// Mitsubishi GX Works2 project: 20151109(M60~65変える前)   PLC: Q03UDV

PROGRAM P1
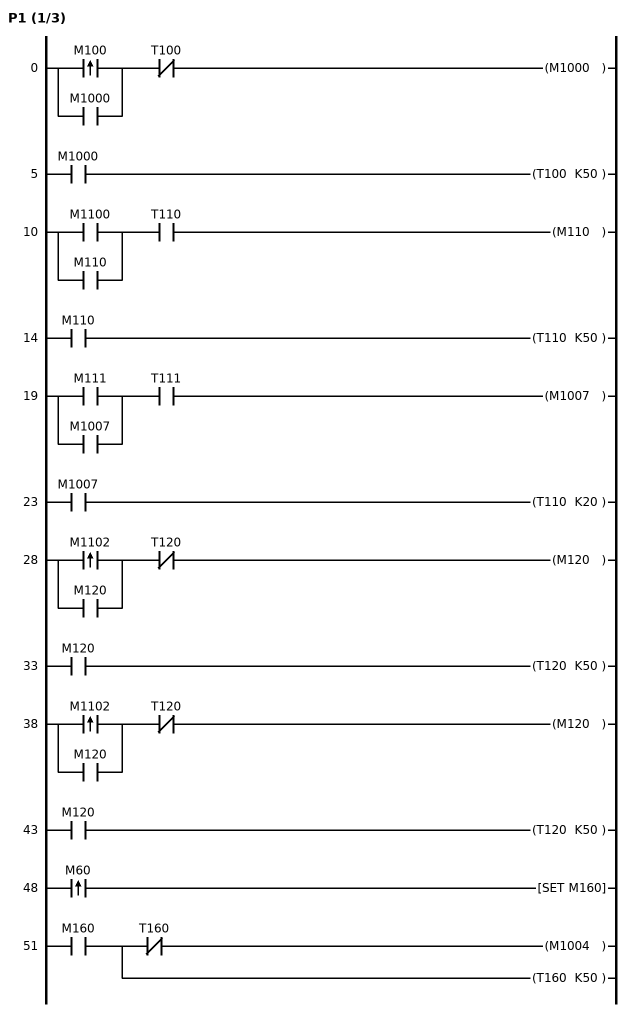
0     LDP     M100
      OR      M1000
      ANI     T100
      OUT     M1000
5     LD      M1000
      OUT     T100 K50
10    LD      M1100
      OR      M110
      AND     T110
      OUT     M110
14    LD      M110
      OUT     T110 K50
19    LD      M111
      OR      M1007
      AND     T111
      OUT     M1007
23    LD      M1007
      OUT     T110 K20
28    LDP     M1102
      OR      M120
      ANI     T120
      OUT     M120
33    LD      M120
      OUT     T120 K50
38    LDP     M1102
      OR      M120
      ANI     T120
      OUT     M120
43    LD      M120
      OUT     T120 K50
48    LDP     M60
      SET     M160
51    LD      M160
      MPS
      ANI     T160
      OUT     M1004
      MPP
      OUT     T160 K50
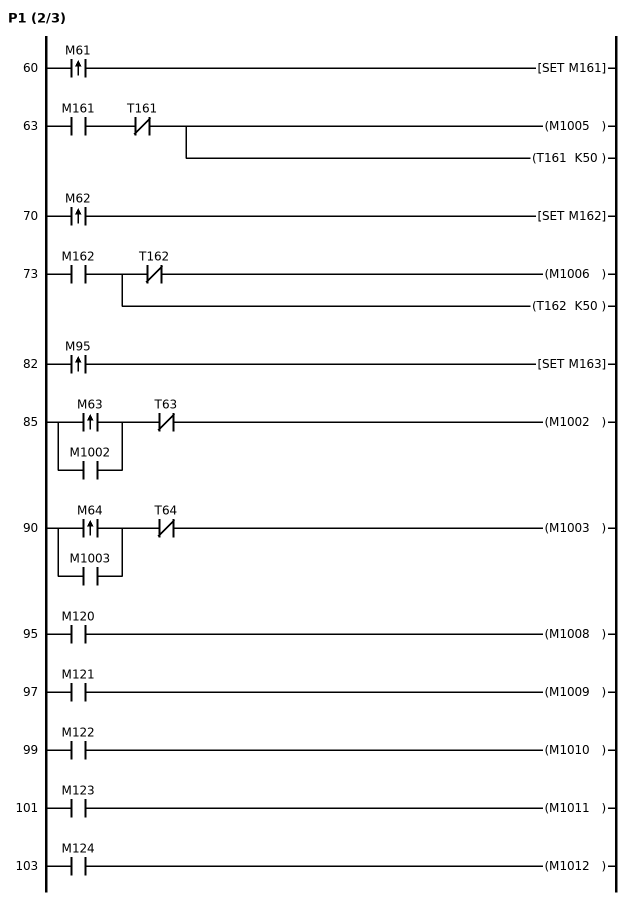
60    LDP     M61
      SET     M161
63    LD      M161
      ANI     T161
      OUT     M1005
      OUT     T161 K50
70    LDP     M62
      SET     M162
73    LD      M162
      MPS
      ANI     T162
      OUT     M1006
      MPP
      OUT     T162 K50
82    LDP     M95
      SET     M163
85    LDP     M63
      OR      M1002
      ANI     T63
      OUT     M1002
90    LDP     M64
      OR      M1003
      ANI     T64
      OUT     M1003
95    LD      M120
      OUT     M1008
97    LD      M121
      OUT     M1009
99    LD      M122
      OUT     M1010
101   LD      M123
      OUT     M1011
103   LD      M124
      OUT     M1012
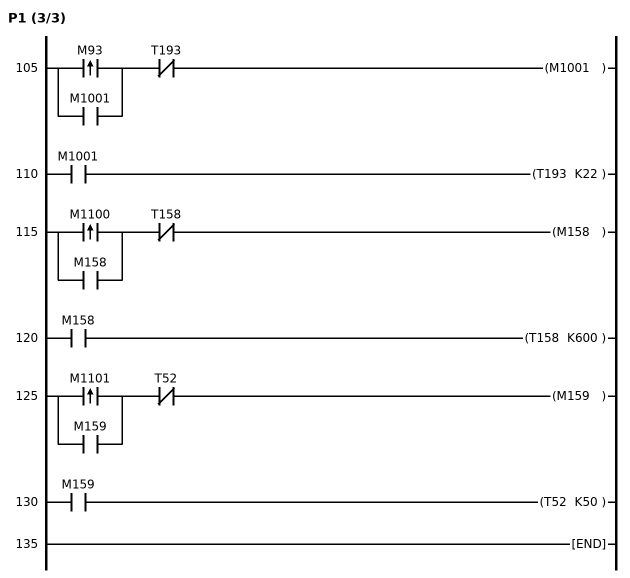
105   LDP     M93
      OR      M1001
      ANI     T193
      OUT     M1001
110   LD      M1001
      OUT     T193 K22
115   LDP     M1100
      OR      M158
      ANI     T158
      OUT     M158
120   LD      M158
      OUT     T158 K600
125   LDP     M1101
      OR      M159
      ANI     T52
      OUT     M159
130   LD      M159
      OUT     T52 K50
135   END
END_PROGRAM

PROGRAM P2
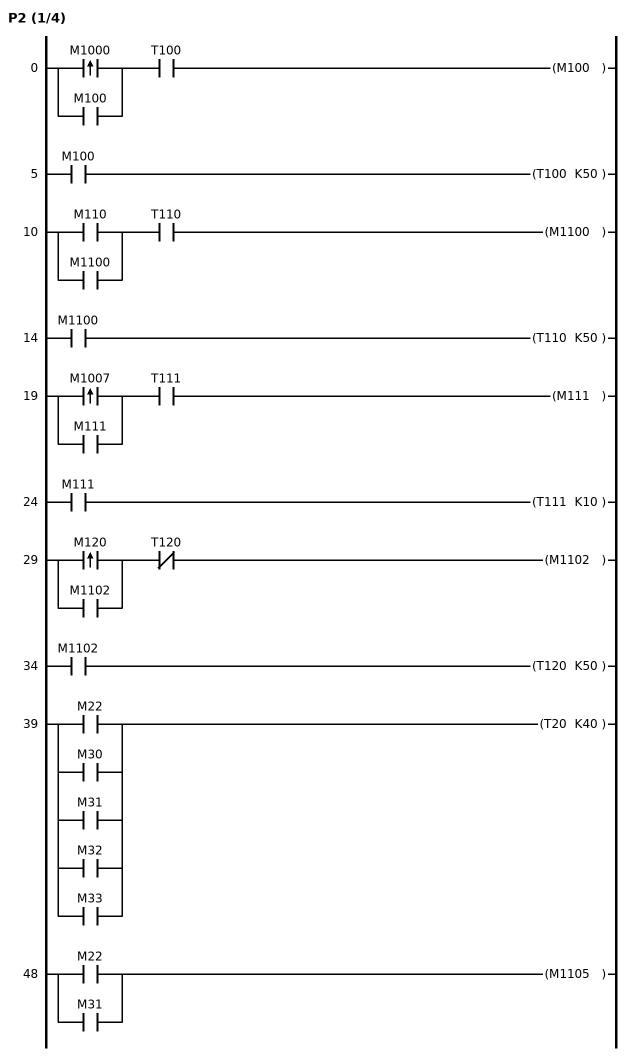
0     LDP     M1000
      OR      M100
      AND     T100
      OUT     M100
5     LD      M100
      OUT     T100 K50
10    LD      M110
      OR      M1100
      AND     T110
      OUT     M1100
14    LD      M1100
      OUT     T110 K50
19    LDP     M1007
      OR      M111
      AND     T111
      OUT     M111
24    LD      M111
      OUT     T111 K10
29    LDP     M120
      OR      M1102
      ANI     T120
      OUT     M1102
34    LD      M1102
      OUT     T120 K50
39    LD      M22
      OR      M30
      OR      M31
      OR      M32
      OR      M33
      OUT     T20 K40
48    LD      M22
      OR      M31
      OUT     M1105
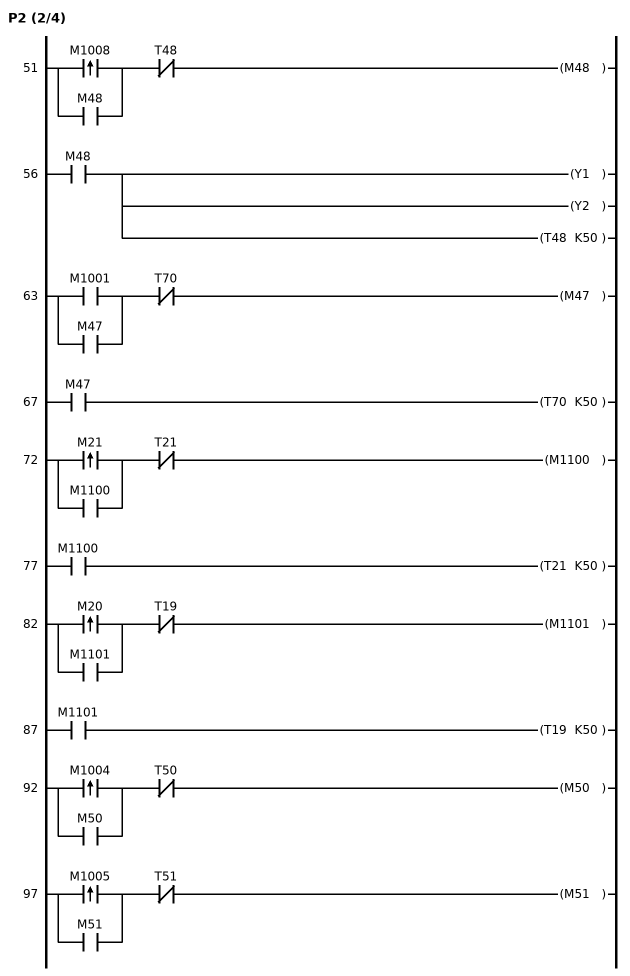
51    LDP     M1008
      OR      M48
      ANI     T48
      OUT     M48
56    LD      M48
      OUT     Y1
      OUT     Y2
      OUT     T48 K50
63    LD      M1001
      OR      M47
      ANI     T70
      OUT     M47
67    LD      M47
      OUT     T70 K50
72    LDP     M21
      OR      M1100
      ANI     T21
      OUT     M1100
77    LD      M1100
      OUT     T21 K50
82    LDP     M20
      OR      M1101
      ANI     T19
      OUT     M1101
87    LD      M1101
      OUT     T19 K50
92    LDP     M1004
      OR      M50
      ANI     T50
      OUT     M50
97    LDP     M1005
      OR      M51
      ANI     T51
      OUT     M51
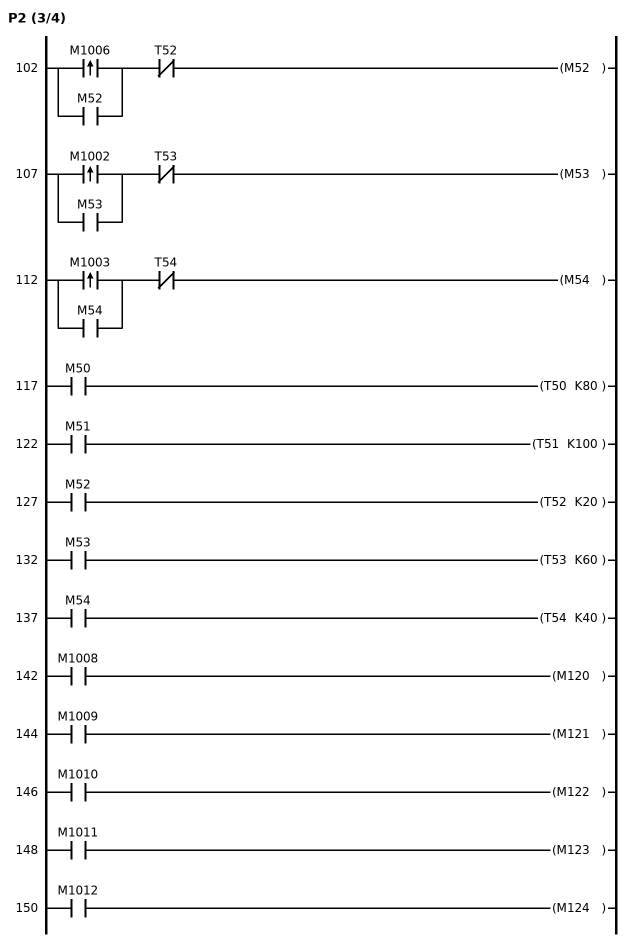
102   LDP     M1006
      OR      M52
      ANI     T52
      OUT     M52
107   LDP     M1002
      OR      M53
      ANI     T53
      OUT     M53
112   LDP     M1003
      OR      M54
      ANI     T54
      OUT     M54
117   LD      M50
      OUT     T50 K80
122   LD      M51
      OUT     T51 K100
127   LD      M52
      OUT     T52 K20
132   LD      M53
      OUT     T53 K60
137   LD      M54
      OUT     T54 K40
142   LD      M1008
      OUT     M120
144   LD      M1009
      OUT     M121
146   LD      M1010
      OUT     M122
148   LD      M1011
      OUT     M123
150   LD      M1012
      OUT     M124
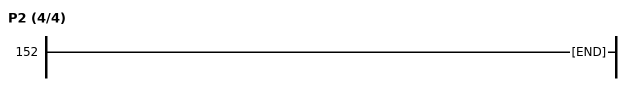
152   END
END_PROGRAM
